(* PLC project Generated.project, CODESYS CODESYS V3.5 SP19 Patch 1 *)
(* stored: creationDateTime 2026-08-18T12:52:51.269652, modificationDateTime 2026-08-18T12:52:51.269652 *)

(* ═══════════════════════════════════════════════════════════════ 🎮 ST_CycleCmd — Commandes IHM pour le cycle semi-automatique ═══════════════════════════════════════════════════════════════ *)
TYPE ST_CycleCmd : STRUCT
  BtnStart : BOOL;  (* ▶️ Lancement cycle automatique *)
  BtnPause : BOOL;  (* ⏸️ Pause cycle automatique *)
  BtnAbort : BOOL;  (* ⏹️ Abandon / arrêt cycle automatique *)
  BtnReset : BOOL;  (* 🔁 Reset dédié FB_Cycle, jamais mélangé au reset défauts général () *)
END_STRUCT;
END_TYPE
